        MoveL Target_3600,v30,fine,DrillTool\WObj:=FakeWing;
SetDO drillDone,1;
WaitUntil drillDone = 0;
        MoveL RelTool(Target_3600,0,0,-10),v30,z10,DrillTool\WObj:=FakeWing;
        MoveL RelTool(Target_3610,0,0,-10),v30,z10,DrillTool\WObj:=FakeWing;
        MoveL Target_3610,v30,fine,DrillTool\WObj:=FakeWing;
SetDO drillDone,1;
WaitUntil drillDone = 0;
        MoveL RelTool(Target_3610,0,0,-10),v30,z10,DrillTool\WObj:=FakeWing;
        MoveL RelTool(Target_3620,0,0,-10),v30,z10,DrillTool\WObj:=FakeWing;
        MoveL Target_3620,v30,fine,DrillTool\WObj:=FakeWing;
SetDO drillDone,1;
WaitUntil drillDone = 0;
        MoveL RelTool(Target_3620,0,0,-10),v30,z10,DrillTool\WObj:=FakeWing;
        MoveL RelTool(Target_3630,0,0,-10),v30,z10,DrillTool\WObj:=FakeWing;
        MoveL Target_3630,v30,fine,DrillTool\WObj:=FakeWing;
SetDO drillDone,1;
WaitUntil drillDone = 0;
        MoveL RelTool(Target_3630,0,0,-10),v30,z10,DrillTool\WObj:=FakeWing;
        MoveL RelTool(Target_3640,0,0,-10),v30,z10,DrillTool\WObj:=FakeWing;
        MoveL Target_3640,v30,fine,DrillTool\WObj:=FakeWing;
SetDO drillDone,1;
WaitUntil drillDone = 0;
        MoveL RelTool(Target_3640,0,0,-10),v30,z10,DrillTool\WObj:=FakeWing;
        MoveL RelTool(Target_3650,0,0,-10),v30,z10,DrillTool\WObj:=FakeWing;
        MoveL Target_3650,v30,fine,DrillTool\WObj:=FakeWing;
SetDO drillDone,1;
WaitUntil drillDone = 0;
        MoveL RelTool(Target_3650,0,0,-10),v30,z10,DrillTool\WObj:=FakeWing;
        MoveL RelTool(Target_3660,0,0,-10),v30,z10,DrillTool\WObj:=FakeWing;
        MoveL Target_3660,v30,fine,DrillTool\WObj:=FakeWing;
SetDO drillDone,1;
WaitUntil drillDone = 0;
        MoveL RelTool(Target_3660,0,0,-10),v30,z10,DrillTool\WObj:=FakeWing;
        MoveL RelTool(Target_3670,0,0,-10),v30,z10,DrillTool\WObj:=FakeWing;
        MoveL Target_3670,v30,fine,DrillTool\WObj:=FakeWing;
SetDO drillDone,1;
WaitUntil drillDone = 0;
        MoveL RelTool(Target_3670,0,0,-10),v30,z10,DrillTool\WObj:=FakeWing;
        MoveL RelTool(Target_3680,0,0,-10),v30,z10,DrillTool\WObj:=FakeWing;
        MoveL Target_3680,v30,fine,DrillTool\WObj:=FakeWing;
SetDO drillDone,1;
WaitUntil drillDone = 0;
        MoveL RelTool(Target_3680,0,0,-10),v30,z10,DrillTool\WObj:=FakeWing;
        MoveL RelTool(Target_3690,0,0,-10),v30,z10,DrillTool\WObj:=FakeWing;
        MoveL Target_3690,v30,fine,DrillTool\WObj:=FakeWing;
SetDO drillDone,1;
WaitUntil drillDone = 0;
        MoveL RelTool(Target_3690,0,0,-10),v30,z10,DrillTool\WObj:=FakeWing;
        MoveL RelTool(Target_3700,0,0,-10),v30,z10,DrillTool\WObj:=FakeWing;
        MoveL Target_3700,v30,fine,DrillTool\WObj:=FakeWing;
SetDO drillDone,1;
WaitUntil drillDone = 0;
        MoveL RelTool(Target_3700,0,0,-10),v30,z10,DrillTool\WObj:=FakeWing;
        MoveL RelTool(Target_3710,0,0,-10),v30,z10,DrillTool\WObj:=FakeWing;
        MoveL Target_3710,v30,fine,DrillTool\WObj:=FakeWing;
SetDO drillDone,1;
WaitUntil drillDone = 0;
        MoveL RelTool(Target_3710,0,0,-10),v30,z10,DrillTool\WObj:=FakeWing;
        MoveL RelTool(Target_3720,0,0,-10),v30,z10,DrillTool\WObj:=FakeWing;
        MoveL Target_3720,v30,fine,DrillTool\WObj:=FakeWing;
SetDO drillDone,1;
WaitUntil drillDone = 0;
        MoveL RelTool(Target_3720,0,0,-10),v30,z10,DrillTool\WObj:=FakeWing;
        MoveL RelTool(Target_3730,0,0,-10),v30,z10,DrillTool\WObj:=FakeWing;
        MoveL Target_3730,v30,fine,DrillTool\WObj:=FakeWing;
SetDO drillDone,1;
WaitUntil drillDone = 0;
        MoveL RelTool(Target_3730,0,0,-10),v30,z10,DrillTool\WObj:=FakeWing;
        MoveL RelTool(Target_3740,0,0,-10),v30,z10,DrillTool\WObj:=FakeWing;
        MoveL Target_3740,v30,fine,DrillTool\WObj:=FakeWing;
SetDO drillDone,1;
WaitUntil drillDone = 0;
        MoveL RelTool(Target_3740,0,0,-10),v30,z10,DrillTool\WObj:=FakeWing;
        MoveL RelTool(Target_3750,0,0,-10),v30,z10,DrillTool\WObj:=FakeWing;
        MoveL Target_3750,v30,fine,DrillTool\WObj:=FakeWing;
SetDO drillDone,1;
WaitUntil drillDone = 0;
        MoveL RelTool(Target_3750,0,0,-10),v30,z10,DrillTool\WObj:=FakeWing;
        MoveL RelTool(Target_3760,0,0,-10),v30,z10,DrillTool\WObj:=FakeWing;
        MoveL Target_3760,v30,fine,DrillTool\WObj:=FakeWing;
SetDO drillDone,1;
WaitUntil drillDone = 0;
        MoveL RelTool(Target_3760,0,0,-10),v30,z10,DrillTool\WObj:=FakeWing;
        MoveL RelTool(Target_3770,0,0,-10),v30,z10,DrillTool\WObj:=FakeWing;
        MoveL Target_3770,v30,fine,DrillTool\WObj:=FakeWing;
SetDO drillDone,1;
WaitUntil drillDone = 0;
        MoveL RelTool(Target_3770,0,0,-10),v30,z10,DrillTool\WObj:=FakeWing;
        MoveL RelTool(Target_3780,0,0,-10),v30,z10,DrillTool\WObj:=FakeWing;
        MoveL Target_3780,v30,fine,DrillTool\WObj:=FakeWing;
SetDO drillDone,1;
WaitUntil drillDone = 0;
        MoveL RelTool(Target_3780,0,0,-10),v30,z10,DrillTool\WObj:=FakeWing;
        MoveL RelTool(Target_3790,0,0,-10),v30,z10,DrillTool\WObj:=FakeWing;
        MoveL Target_3790,v30,fine,DrillTool\WObj:=FakeWing;
SetDO drillDone,1;
WaitUntil drillDone = 0;
        MoveL RelTool(Target_3790,0,0,-10),v30,z10,DrillTool\WObj:=FakeWing;
        MoveL RelTool(Target_3800,0,0,-10),v30,z10,DrillTool\WObj:=FakeWing;
        MoveL Target_3800,v30,fine,DrillTool\WObj:=FakeWing;
SetDO drillDone,1;
WaitUntil drillDone = 0;
        MoveL RelTool(Target_3800,0,0,-10),v30,z10,DrillTool\WObj:=FakeWing;
        MoveL RelTool(Target_3810,0,0,-10),v30,z10,DrillTool\WObj:=FakeWing;
        MoveL Target_3810,v30,fine,DrillTool\WObj:=FakeWing;
SetDO drillDone,1;
WaitUntil drillDone = 0;
        MoveL RelTool(Target_3810,0,0,-10),v30,z10,DrillTool\WObj:=FakeWing;
        MoveL RelTool(Target_3820,0,0,-10),v30,z10,DrillTool\WObj:=FakeWing;
        MoveL Target_3820,v30,fine,DrillTool\WObj:=FakeWing;
SetDO drillDone,1;
WaitUntil drillDone = 0;
        MoveL RelTool(Target_3820,0,0,-10),v30,z10,DrillTool\WObj:=FakeWing;
        MoveL RelTool(Target_3830,0,0,-10),v30,z10,DrillTool\WObj:=FakeWing;
        MoveL Target_3830,v30,fine,DrillTool\WObj:=FakeWing;
SetDO drillDone,1;
WaitUntil drillDone = 0;
        MoveL RelTool(Target_3830,0,0,-10),v30,z10,DrillTool\WObj:=FakeWing;
        MoveL RelTool(Target_3840,0,0,-10),v30,z10,DrillTool\WObj:=FakeWing;
        MoveL Target_3840,v30,fine,DrillTool\WObj:=FakeWing;
SetDO drillDone,1;
WaitUntil drillDone = 0;
        MoveL RelTool(Target_3840,0,0,-10),v30,z10,DrillTool\WObj:=FakeWing;
        MoveL RelTool(Target_3850,0,0,-10),v30,z10,DrillTool\WObj:=FakeWing;
        MoveL Target_3850,v30,fine,DrillTool\WObj:=FakeWing;
SetDO drillDone,1;
WaitUntil drillDone = 0;
        MoveL RelTool(Target_3850,0,0,-10),v30,z10,DrillTool\WObj:=FakeWing;
        MoveL RelTool(Target_3860,0,0,-10),v30,z10,DrillTool\WObj:=FakeWing;
        MoveL Target_3860,v30,fine,DrillTool\WObj:=FakeWing;
SetDO drillDone,1;
WaitUntil drillDone = 0;
        MoveL RelTool(Target_3860,0,0,-10),v30,z10,DrillTool\WObj:=FakeWing;
        MoveL RelTool(Target_3870,0,0,-10),v30,z10,DrillTool\WObj:=FakeWing;
        MoveL Target_3870,v30,fine,DrillTool\WObj:=FakeWing;
SetDO drillDone,1;
WaitUntil drillDone = 0;
        MoveL RelTool(Target_3870,0,0,-10),v30,z10,DrillTool\WObj:=FakeWing;
        MoveL RelTool(Target_3880,0,0,-10),v30,z10,DrillTool\WObj:=FakeWing;
        MoveL Target_3880,v30,fine,DrillTool\WObj:=FakeWing;
SetDO drillDone,1;
WaitUntil drillDone = 0;
        MoveL RelTool(Target_3880,0,0,-10),v30,z10,DrillTool\WObj:=FakeWing;
        MoveL RelTool(Target_3890,0,0,-10),v30,z10,DrillTool\WObj:=FakeWing;
        MoveL Target_3890,v30,fine,DrillTool\WObj:=FakeWing;
SetDO drillDone,1;
WaitUntil drillDone = 0;
        MoveL RelTool(Target_3890,0,0,-10),v30,z10,DrillTool\WObj:=FakeWing;
        MoveL RelTool(Target_3900,0,0,-10),v30,z10,DrillTool\WObj:=FakeWing;
        MoveL Target_3900,v30,fine,DrillTool\WObj:=FakeWing;
SetDO drillDone,1;
WaitUntil drillDone = 0;
        MoveL RelTool(Target_3900,0,0,-10),v30,z10,DrillTool\WObj:=FakeWing;
        MoveL RelTool(Target_3910,0,0,-10),v30,z10,DrillTool\WObj:=FakeWing;
        MoveL Target_3910,v30,fine,DrillTool\WObj:=FakeWing;
SetDO drillDone,1;
WaitUntil drillDone = 0;
        MoveL RelTool(Target_3910,0,0,-10),v30,z10,DrillTool\WObj:=FakeWing;
        MoveL RelTool(Target_3920,0,0,-10),v30,z10,DrillTool\WObj:=FakeWing;
        MoveL Target_3920,v30,fine,DrillTool\WObj:=FakeWing;
SetDO drillDone,1;
WaitUntil drillDone = 0;
        MoveL RelTool(Target_3920,0,0,-10),v30,z10,DrillTool\WObj:=FakeWing;
        MoveL RelTool(Target_3930,0,0,-10),v30,z10,DrillTool\WObj:=FakeWing;
        MoveL Target_3930,v30,fine,DrillTool\WObj:=FakeWing;
SetDO drillDone,1;
WaitUntil drillDone = 0;
        MoveL RelTool(Target_3930,0,0,-10),v30,z10,DrillTool\WObj:=FakeWing;
        MoveL RelTool(Target_3940,0,0,-10),v30,z10,DrillTool\WObj:=FakeWing;
        MoveL Target_3940,v30,fine,DrillTool\WObj:=FakeWing;
SetDO drillDone,1;
WaitUntil drillDone = 0;
        MoveL RelTool(Target_3940,0,0,-10),v30,z10,DrillTool\WObj:=FakeWing;
        MoveL RelTool(Target_3950,0,0,-10),v30,z10,DrillTool\WObj:=FakeWing;
        MoveL Target_3950,v30,fine,DrillTool\WObj:=FakeWing;
SetDO drillDone,1;
WaitUntil drillDone = 0;
        MoveL RelTool(Target_3950,0,0,-10),v30,z10,DrillTool\WObj:=FakeWing;
        MoveL RelTool(Target_3960,0,0,-10),v30,z10,DrillTool\WObj:=FakeWing;
        MoveL Target_3960,v30,fine,DrillTool\WObj:=FakeWing;
SetDO drillDone,1;
WaitUntil drillDone = 0;
        MoveL RelTool(Target_3960,0,0,-10),v30,z10,DrillTool\WObj:=FakeWing;
        MoveL RelTool(Target_3970,0,0,-10),v30,z10,DrillTool\WObj:=FakeWing;
        MoveL Target_3970,v30,fine,DrillTool\WObj:=FakeWing;
SetDO drillDone,1;
WaitUntil drillDone = 0;
        MoveL RelTool(Target_3970,0,0,-10),v30,z10,DrillTool\WObj:=FakeWing;
        MoveL RelTool(Target_3980,0,0,-10),v30,z10,DrillTool\WObj:=FakeWing;
        MoveL Target_3980,v30,fine,DrillTool\WObj:=FakeWing;
SetDO drillDone,1;
WaitUntil drillDone = 0;
        MoveL RelTool(Target_3980,0,0,-10),v30,z10,DrillTool\WObj:=FakeWing;
        MoveL RelTool(Target_3990,0,0,-10),v30,z10,DrillTool\WObj:=FakeWing;
        MoveL Target_3990,v30,fine,DrillTool\WObj:=FakeWing;
SetDO drillDone,1;
WaitUntil drillDone = 0;
        MoveL RelTool(Target_3990,0,0,-10),v30,z10,DrillTool\WObj:=FakeWing;
        MoveL RelTool(Target_4000,0,0,-10),v30,z10,DrillTool\WObj:=FakeWing;
        MoveL Target_4000,v30,fine,DrillTool\WObj:=FakeWing;
SetDO drillDone,1;
WaitUntil drillDone = 0;
        MoveL RelTool(Target_4000,0,0,-10),v30,z10,DrillTool\WObj:=FakeWing;
        MoveL RelTool(Target_4010,0,0,-10),v30,z10,DrillTool\WObj:=FakeWing;
        MoveL Target_4010,v30,fine,DrillTool\WObj:=FakeWing;
SetDO drillDone,1;
WaitUntil drillDone = 0;
        MoveL RelTool(Target_4010,0,0,-10),v30,z10,DrillTool\WObj:=FakeWing;
        MoveL RelTool(Target_4020,0,0,-10),v30,z10,DrillTool\WObj:=FakeWing;
        MoveL Target_4020,v30,fine,DrillTool\WObj:=FakeWing;
SetDO drillDone,1;
WaitUntil drillDone = 0;
        MoveL RelTool(Target_4020,0,0,-10),v30,z10,DrillTool\WObj:=FakeWing;
        MoveL RelTool(Target_4030,0,0,-10),v30,z10,DrillTool\WObj:=FakeWing;
        MoveL Target_4030,v30,fine,DrillTool\WObj:=FakeWing;
SetDO drillDone,1;
WaitUntil drillDone = 0;
        MoveL RelTool(Target_4030,0,0,-10),v30,z10,DrillTool\WObj:=FakeWing;
        MoveL RelTool(Target_4040,0,0,-10),v30,z10,DrillTool\WObj:=FakeWing;
        MoveL Target_4040,v30,fine,DrillTool\WObj:=FakeWing;
SetDO drillDone,1;
WaitUntil drillDone = 0;
        MoveL RelTool(Target_4040,0,0,-10),v30,z10,DrillTool\WObj:=FakeWing;
        MoveL RelTool(Target_4050,0,0,-10),v30,z10,DrillTool\WObj:=FakeWing;
        MoveL Target_4050,v30,fine,DrillTool\WObj:=FakeWing;
SetDO drillDone,1;
WaitUntil drillDone = 0;
        MoveL RelTool(Target_4050,0,0,-10),v30,z10,DrillTool\WObj:=FakeWing;
        MoveL RelTool(Target_4060,0,0,-10),v30,z10,DrillTool\WObj:=FakeWing;
        MoveL Target_4060,v30,fine,DrillTool\WObj:=FakeWing;
SetDO drillDone,1;
WaitUntil drillDone = 0;
        MoveL RelTool(Target_4060,0,0,-10),v30,z10,DrillTool\WObj:=FakeWing;
        MoveL RelTool(Target_4070,0,0,-10),v30,z10,DrillTool\WObj:=FakeWing;
        MoveL Target_4070,v30,fine,DrillTool\WObj:=FakeWing;
SetDO drillDone,1;
WaitUntil drillDone = 0;
        MoveL RelTool(Target_4070,0,0,-10),v30,z10,DrillTool\WObj:=FakeWing;
        MoveL RelTool(Target_4080,0,0,-10),v30,z10,DrillTool\WObj:=FakeWing;
        MoveL Target_4080,v30,fine,DrillTool\WObj:=FakeWing;
SetDO drillDone,1;
WaitUntil drillDone = 0;
        MoveL RelTool(Target_4080,0,0,-10),v30,z10,DrillTool\WObj:=FakeWing;
        MoveL RelTool(Target_4090,0,0,-10),v30,z10,DrillTool\WObj:=FakeWing;
        MoveL Target_4090,v30,fine,DrillTool\WObj:=FakeWing;
SetDO drillDone,1;
WaitUntil drillDone = 0;
        MoveL RelTool(Target_4090,0,0,-10),v30,z10,DrillTool\WObj:=FakeWing;
        MoveL RelTool(Target_4100,0,0,-10),v30,z10,DrillTool\WObj:=FakeWing;
        MoveL Target_4100,v30,fine,DrillTool\WObj:=FakeWing;
SetDO drillDone,1;
WaitUntil drillDone = 0;
        MoveL RelTool(Target_4100,0,0,-10),v30,z10,DrillTool\WObj:=FakeWing;
        MoveL RelTool(Target_4110,0,0,-10),v30,z10,DrillTool\WObj:=FakeWing;
        MoveL Target_4110,v30,fine,DrillTool\WObj:=FakeWing;
SetDO drillDone,1;
WaitUntil drillDone = 0;
        MoveL RelTool(Target_4110,0,0,-10),v30,z10,DrillTool\WObj:=FakeWing;
        MoveL RelTool(Target_4120,0,0,-10),v30,z10,DrillTool\WObj:=FakeWing;
        MoveL Target_4120,v30,fine,DrillTool\WObj:=FakeWing;
SetDO drillDone,1;
WaitUntil drillDone = 0;
        MoveL RelTool(Target_4120,0,0,-10),v30,z10,DrillTool\WObj:=FakeWing;
        MoveL RelTool(Target_4130,0,0,-10),v30,z10,DrillTool\WObj:=FakeWing;
        MoveL Target_4130,v30,fine,DrillTool\WObj:=FakeWing;
SetDO drillDone,1;
WaitUntil drillDone = 0;
        MoveL RelTool(Target_4130,0,0,-10),v30,z10,DrillTool\WObj:=FakeWing;
        MoveL RelTool(Target_4140,0,0,-10),v30,z10,DrillTool\WObj:=FakeWing;
        MoveL Target_4140,v30,fine,DrillTool\WObj:=FakeWing;
SetDO drillDone,1;
WaitUntil drillDone = 0;
        MoveL RelTool(Target_4140,0,0,-10),v30,z10,DrillTool\WObj:=FakeWing;
        MoveL RelTool(Target_4150,0,0,-10),v30,z10,DrillTool\WObj:=FakeWing;
        MoveL Target_4150,v30,fine,DrillTool\WObj:=FakeWing;
SetDO drillDone,1;
WaitUntil drillDone = 0;
        MoveL RelTool(Target_4150,0,0,-10),v30,z10,DrillTool\WObj:=FakeWing;
        MoveL RelTool(Target_4160,0,0,-10),v30,z10,DrillTool\WObj:=FakeWing;
        MoveL Target_4160,v30,fine,DrillTool\WObj:=FakeWing;
SetDO drillDone,1;
WaitUntil drillDone = 0;
        MoveL RelTool(Target_4160,0,0,-10),v30,z10,DrillTool\WObj:=FakeWing;
        MoveL RelTool(Target_4170,0,0,-10),v30,z10,DrillTool\WObj:=FakeWing;
        MoveL Target_4170,v30,fine,DrillTool\WObj:=FakeWing;
SetDO drillDone,1;
WaitUntil drillDone = 0;
        MoveL RelTool(Target_4170,0,0,-10),v30,z10,DrillTool\WObj:=FakeWing;
        MoveL RelTool(Target_4180,0,0,-10),v30,z10,DrillTool\WObj:=FakeWing;
        MoveL Target_4180,v30,fine,DrillTool\WObj:=FakeWing;
SetDO drillDone,1;
WaitUntil drillDone = 0;
        MoveL RelTool(Target_4180,0,0,-10),v30,z10,DrillTool\WObj:=FakeWing;
        MoveL RelTool(Target_4190,0,0,-10),v30,z10,DrillTool\WObj:=FakeWing;
        MoveL Target_4190,v30,fine,DrillTool\WObj:=FakeWing;
SetDO drillDone,1;
WaitUntil drillDone = 0;
        MoveL RelTool(Target_4190,0,0,-10),v30,z10,DrillTool\WObj:=FakeWing;
        MoveL RelTool(Target_4200,0,0,-10),v30,z10,DrillTool\WObj:=FakeWing;
        MoveL Target_4200,v30,fine,DrillTool\WObj:=FakeWing;
SetDO drillDone,1;
WaitUntil drillDone = 0;
        MoveL RelTool(Target_4200,0,0,-10),v30,z10,DrillTool\WObj:=FakeWing;
        MoveL RelTool(Target_4210,0,0,-10),v30,z10,DrillTool\WObj:=FakeWing;
        MoveL Target_4210,v30,fine,DrillTool\WObj:=FakeWing;
SetDO drillDone,1;
WaitUntil drillDone = 0;
        MoveL RelTool(Target_4210,0,0,-10),v30,z10,DrillTool\WObj:=FakeWing;
        MoveL RelTool(Target_4220,0,0,-10),v30,z10,DrillTool\WObj:=FakeWing;
        MoveL Target_4220,v30,fine,DrillTool\WObj:=FakeWing;
SetDO drillDone,1;
WaitUntil drillDone = 0;
        MoveL RelTool(Target_4220,0,0,-10),v30,z10,DrillTool\WObj:=FakeWing;
        MoveL RelTool(Target_4230,0,0,-10),v30,z10,DrillTool\WObj:=FakeWing;
        MoveL Target_4230,v30,fine,DrillTool\WObj:=FakeWing;
SetDO drillDone,1;
WaitUntil drillDone = 0;
        MoveL RelTool(Target_4230,0,0,-10),v30,z10,DrillTool\WObj:=FakeWing;
        MoveL RelTool(Target_4240,0,0,-10),v30,z10,DrillTool\WObj:=FakeWing;
        MoveL Target_4240,v30,fine,DrillTool\WObj:=FakeWing;
SetDO drillDone,1;
WaitUntil drillDone = 0;
        MoveL RelTool(Target_4240,0,0,-10),v30,z10,DrillTool\WObj:=FakeWing;
        MoveL RelTool(Target_4250,0,0,-10),v30,z10,DrillTool\WObj:=FakeWing;
        MoveL Target_4250,v30,fine,DrillTool\WObj:=FakeWing;
SetDO drillDone,1;
WaitUntil drillDone = 0;
        MoveL RelTool(Target_4250,0,0,-10),v30,z10,DrillTool\WObj:=FakeWing;
        MoveL RelTool(Target_4260,0,0,-10),v30,z10,DrillTool\WObj:=FakeWing;
        MoveL Target_4260,v30,fine,DrillTool\WObj:=FakeWing;
SetDO drillDone,1;
WaitUntil drillDone = 0;
        MoveL RelTool(Target_4260,0,0,-10),v30,z10,DrillTool\WObj:=FakeWing;
        MoveL RelTool(Target_4270,0,0,-10),v30,z10,DrillTool\WObj:=FakeWing;
        MoveL Target_4270,v30,fine,DrillTool\WObj:=FakeWing;
SetDO drillDone,1;
WaitUntil drillDone = 0;
        MoveL RelTool(Target_4270,0,0,-10),v30,z10,DrillTool\WObj:=FakeWing;
        MoveL RelTool(Target_4280,0,0,-10),v30,z10,DrillTool\WObj:=FakeWing;
        MoveL Target_4280,v30,fine,DrillTool\WObj:=FakeWing;
SetDO drillDone,1;
WaitUntil drillDone = 0;
        MoveL RelTool(Target_4280,0,0,-10),v30,z10,DrillTool\WObj:=FakeWing;
        MoveL RelTool(Target_4290,0,0,-10),v30,z10,DrillTool\WObj:=FakeWing;
        MoveL Target_4290,v30,fine,DrillTool\WObj:=FakeWing;
SetDO drillDone,1;
WaitUntil drillDone = 0;
        MoveL RelTool(Target_4290,0,0,-10),v30,z10,DrillTool\WObj:=FakeWing;
        MoveL RelTool(Target_4300,0,0,-10),v30,z10,DrillTool\WObj:=FakeWing;
        MoveL Target_4300,v30,fine,DrillTool\WObj:=FakeWing;
SetDO drillDone,1;
WaitUntil drillDone = 0;
        MoveL RelTool(Target_4300,0,0,-10),v30,z10,DrillTool\WObj:=FakeWing;
        MoveL RelTool(Target_4310,0,0,-10),v30,z10,DrillTool\WObj:=FakeWing;
        MoveL Target_4310,v30,fine,DrillTool\WObj:=FakeWing;
SetDO drillDone,1;
WaitUntil drillDone = 0;
        MoveL RelTool(Target_4310,0,0,-10),v30,z10,DrillTool\WObj:=FakeWing;
        MoveL RelTool(Target_4320,0,0,-10),v30,z10,DrillTool\WObj:=FakeWing;
        MoveL Target_4320,v30,fine,DrillTool\WObj:=FakeWing;
SetDO drillDone,1;
WaitUntil drillDone = 0;
        MoveL RelTool(Target_4320,0,0,-10),v30,z10,DrillTool\WObj:=FakeWing;
        MoveL RelTool(Target_4330,0,0,-10),v30,z10,DrillTool\WObj:=FakeWing;
        MoveL Target_4330,v30,fine,DrillTool\WObj:=FakeWing;
SetDO drillDone,1;
WaitUntil drillDone = 0;
        MoveL RelTool(Target_4330,0,0,-10),v30,z10,DrillTool\WObj:=FakeWing;
        MoveL RelTool(Target_4340,0,0,-10),v30,z10,DrillTool\WObj:=FakeWing;
        MoveL Target_4340,v30,fine,DrillTool\WObj:=FakeWing;
SetDO drillDone,1;
WaitUntil drillDone = 0;
        MoveL RelTool(Target_4340,0,0,-10),v30,z10,DrillTool\WObj:=FakeWing;
        MoveL RelTool(Target_4350,0,0,-10),v30,z10,DrillTool\WObj:=FakeWing;
        MoveL Target_4350,v30,fine,DrillTool\WObj:=FakeWing;
SetDO drillDone,1;
WaitUntil drillDone = 0;
        MoveL RelTool(Target_4350,0,0,-10),v30,z10,DrillTool\WObj:=FakeWing;
        MoveL RelTool(Target_4360,0,0,-10),v30,z10,DrillTool\WObj:=FakeWing;
        MoveL Target_4360,v30,fine,DrillTool\WObj:=FakeWing;
SetDO drillDone,1;
WaitUntil drillDone = 0;
        MoveL RelTool(Target_4360,0,0,-10),v30,z10,DrillTool\WObj:=FakeWing;
        MoveL RelTool(Target_4370,0,0,-10),v30,z10,DrillTool\WObj:=FakeWing;
        MoveL Target_4370,v30,fine,DrillTool\WObj:=FakeWing;
SetDO drillDone,1;
WaitUntil drillDone = 0;
        MoveL RelTool(Target_4370,0,0,-10),v30,z10,DrillTool\WObj:=FakeWing;
        MoveL RelTool(Target_4380,0,0,-10),v30,z10,DrillTool\WObj:=FakeWing;
        MoveL Target_4380,v30,fine,DrillTool\WObj:=FakeWing;
SetDO drillDone,1;
WaitUntil drillDone = 0;
        MoveL RelTool(Target_4380,0,0,-10),v30,z10,DrillTool\WObj:=FakeWing;
        MoveL RelTool(Target_4390,0,0,-10),v30,z10,DrillTool\WObj:=FakeWing;
        MoveL Target_4390,v30,fine,DrillTool\WObj:=FakeWing;
SetDO drillDone,1;
WaitUntil drillDone = 0;
        MoveL RelTool(Target_4390,0,0,-10),v30,z10,DrillTool\WObj:=FakeWing;
        MoveL RelTool(Target_4400,0,0,-10),v30,z10,DrillTool\WObj:=FakeWing;
        MoveL Target_4400,v30,fine,DrillTool\WObj:=FakeWing;
SetDO drillDone,1;
WaitUntil drillDone = 0;
        MoveL RelTool(Target_4400,0,0,-10),v30,z10,DrillTool\WObj:=FakeWing;
        MoveL RelTool(Target_4410,0,0,-10),v30,z10,DrillTool\WObj:=FakeWing;
        MoveL Target_4410,v30,fine,DrillTool\WObj:=FakeWing;
SetDO drillDone,1;
WaitUntil drillDone = 0;
        MoveL RelTool(Target_4410,0,0,-10),v30,z10,DrillTool\WObj:=FakeWing;
        MoveL RelTool(Target_4420,0,0,-10),v30,z10,DrillTool\WObj:=FakeWing;
        MoveL Target_4420,v30,fine,DrillTool\WObj:=FakeWing;
SetDO drillDone,1;
WaitUntil drillDone = 0;
        MoveL RelTool(Target_4420,0,0,-10),v30,z10,DrillTool\WObj:=FakeWing;
        MoveL RelTool(Target_4430,0,0,-10),v30,z10,DrillTool\WObj:=FakeWing;
        MoveL Target_4430,v30,fine,DrillTool\WObj:=FakeWing;
SetDO drillDone,1;
WaitUntil drillDone = 0;
        MoveL RelTool(Target_4430,0,0,-10),v30,z10,DrillTool\WObj:=FakeWing;
        MoveL RelTool(Target_4440,0,0,-10),v30,z10,DrillTool\WObj:=FakeWing;
        MoveL Target_4440,v30,fine,DrillTool\WObj:=FakeWing;
SetDO drillDone,1;
WaitUntil drillDone = 0;
        MoveL RelTool(Target_4440,0,0,-10),v30,z10,DrillTool\WObj:=FakeWing;
        MoveL RelTool(Target_4450,0,0,-10),v30,z10,DrillTool\WObj:=FakeWing;
        MoveL Target_4450,v30,fine,DrillTool\WObj:=FakeWing;
SetDO drillDone,1;
WaitUntil drillDone = 0;
        MoveL RelTool(Target_4450,0,0,-10),v30,z10,DrillTool\WObj:=FakeWing;
        MoveL RelTool(Target_4460,0,0,-10),v30,z10,DrillTool\WObj:=FakeWing;
        MoveL Target_4460,v30,fine,DrillTool\WObj:=FakeWing;
SetDO drillDone,1;
WaitUntil drillDone = 0;
        MoveL RelTool(Target_4460,0,0,-10),v30,z10,DrillTool\WObj:=FakeWing;
        MoveL RelTool(Target_4470,0,0,-10),v30,z10,DrillTool\WObj:=FakeWing;
        MoveL Target_4470,v30,fine,DrillTool\WObj:=FakeWing;
SetDO drillDone,1;
WaitUntil drillDone = 0;
        MoveL RelTool(Target_4470,0,0,-10),v30,z10,DrillTool\WObj:=FakeWing;
        MoveL RelTool(Target_4480,0,0,-10),v30,z10,DrillTool\WObj:=FakeWing;
        MoveL Target_4480,v30,fine,DrillTool\WObj:=FakeWing;
SetDO drillDone,1;
WaitUntil drillDone = 0;
        MoveL RelTool(Target_4480,0,0,-10),v30,z10,DrillTool\WObj:=FakeWing;
        MoveL RelTool(Target_4490,0,0,-10),v30,z10,DrillTool\WObj:=FakeWing;
        MoveL Target_4490,v30,fine,DrillTool\WObj:=FakeWing;
SetDO drillDone,1;
WaitUntil drillDone = 0;
        MoveL RelTool(Target_4490,0,0,-10),v30,z10,DrillTool\WObj:=FakeWing;
        MoveL RelTool(Target_4500,0,0,-10),v30,z10,DrillTool\WObj:=FakeWing;
        MoveL Target_4500,v30,fine,DrillTool\WObj:=FakeWing;
SetDO drillDone,1;
WaitUntil drillDone = 0;
        MoveL RelTool(Target_4500,0,0,-10),v30,z10,DrillTool\WObj:=FakeWing;
        MoveL RelTool(Target_4510,0,0,-10),v30,z10,DrillTool\WObj:=FakeWing;
        MoveL Target_4510,v30,fine,DrillTool\WObj:=FakeWing;
SetDO drillDone,1;
WaitUntil drillDone = 0;
        MoveL RelTool(Target_4510,0,0,-10),v30,z10,DrillTool\WObj:=FakeWing;
        MoveL RelTool(Target_4520,0,0,-10),v30,z10,DrillTool\WObj:=FakeWing;
        MoveL Target_4520,v30,fine,DrillTool\WObj:=FakeWing;
SetDO drillDone,1;
WaitUntil drillDone = 0;
        MoveL RelTool(Target_4520,0,0,-10),v30,z10,DrillTool\WObj:=FakeWing;
        MoveL RelTool(Target_4530,0,0,-10),v30,z10,DrillTool\WObj:=FakeWing;
        MoveL Target_4530,v30,fine,DrillTool\WObj:=FakeWing;
SetDO drillDone,1;
WaitUntil drillDone = 0;
        MoveL RelTool(Target_4530,0,0,-10),v30,z10,DrillTool\WObj:=FakeWing;
        MoveL RelTool(Target_4540,0,0,-10),v30,z10,DrillTool\WObj:=FakeWing;
        MoveL Target_4540,v30,fine,DrillTool\WObj:=FakeWing;
SetDO drillDone,1;
WaitUntil drillDone = 0;
        MoveL RelTool(Target_4540,0,0,-10),v30,z10,DrillTool\WObj:=FakeWing;
        MoveL RelTool(Target_4550,0,0,-10),v30,z10,DrillTool\WObj:=FakeWing;
        MoveL Target_4550,v30,fine,DrillTool\WObj:=FakeWing;
SetDO drillDone,1;
WaitUntil drillDone = 0;
        MoveL RelTool(Target_4550,0,0,-10),v30,z10,DrillTool\WObj:=FakeWing;
        MoveL RelTool(Target_4560,0,0,-10),v30,z10,DrillTool\WObj:=FakeWing;
        MoveL Target_4560,v30,fine,DrillTool\WObj:=FakeWing;
SetDO drillDone,1;
WaitUntil drillDone = 0;
        MoveL RelTool(Target_4560,0,0,-10),v30,z10,DrillTool\WObj:=FakeWing;
        MoveL RelTool(Target_4570,0,0,-10),v30,z10,DrillTool\WObj:=FakeWing;
        MoveL Target_4570,v30,fine,DrillTool\WObj:=FakeWing;
SetDO drillDone,1;
WaitUntil drillDone = 0;
        MoveL RelTool(Target_4570,0,0,-10),v30,z10,DrillTool\WObj:=FakeWing;
        MoveL RelTool(Target_4580,0,0,-10),v30,z10,DrillTool\WObj:=FakeWing;
        MoveL Target_4580,v30,fine,DrillTool\WObj:=FakeWing;
SetDO drillDone,1;
WaitUntil drillDone = 0;
        MoveL RelTool(Target_4580,0,0,-10),v30,z10,DrillTool\WObj:=FakeWing;
        MoveL RelTool(Target_4590,0,0,-10),v30,z10,DrillTool\WObj:=FakeWing;
        MoveL Target_4590,v30,fine,DrillTool\WObj:=FakeWing;
SetDO drillDone,1;
WaitUntil drillDone = 0;
        MoveL RelTool(Target_4590,0,0,-10),v30,z10,DrillTool\WObj:=FakeWing;
        MoveL RelTool(Target_4600,0,0,-10),v30,z10,DrillTool\WObj:=FakeWing;
        MoveL Target_4600,v30,fine,DrillTool\WObj:=FakeWing;
SetDO drillDone,1;
WaitUntil drillDone = 0;
        MoveL RelTool(Target_4600,0,0,-10),v30,z10,DrillTool\WObj:=FakeWing;
        MoveL RelTool(Target_4610,0,0,-10),v30,z10,DrillTool\WObj:=FakeWing;
        MoveL Target_4610,v30,fine,DrillTool\WObj:=FakeWing;
SetDO drillDone,1;
WaitUntil drillDone = 0;
        MoveL RelTool(Target_4610,0,0,-10),v30,z10,DrillTool\WObj:=FakeWing;
        MoveL RelTool(Target_4620,0,0,-10),v30,z10,DrillTool\WObj:=FakeWing;
        MoveL Target_4620,v30,fine,DrillTool\WObj:=FakeWing;
SetDO drillDone,1;
WaitUntil drillDone = 0;
        MoveL RelTool(Target_4620,0,0,-10),v30,z10,DrillTool\WObj:=FakeWing;
        MoveL RelTool(Target_4630,0,0,-10),v30,z10,DrillTool\WObj:=FakeWing;
        MoveL Target_4630,v30,fine,DrillTool\WObj:=FakeWing;
SetDO drillDone,1;
WaitUntil drillDone = 0;
        MoveL RelTool(Target_4630,0,0,-10),v30,z10,DrillTool\WObj:=FakeWing;
        MoveL RelTool(Target_4640,0,0,-10),v30,z10,DrillTool\WObj:=FakeWing;
        MoveL Target_4640,v30,fine,DrillTool\WObj:=FakeWing;
SetDO drillDone,1;
WaitUntil drillDone = 0;
        MoveL RelTool(Target_4640,0,0,-10),v30,z10,DrillTool\WObj:=FakeWing;
        MoveL RelTool(Target_4650,0,0,-10),v30,z10,DrillTool\WObj:=FakeWing;
        MoveL Target_4650,v30,fine,DrillTool\WObj:=FakeWing;
SetDO drillDone,1;
WaitUntil drillDone = 0;
        MoveL RelTool(Target_4650,0,0,-10),v30,z10,DrillTool\WObj:=FakeWing;
        MoveL RelTool(Target_4660,0,0,-10),v30,z10,DrillTool\WObj:=FakeWing;
        MoveL Target_4660,v30,fine,DrillTool\WObj:=FakeWing;
SetDO drillDone,1;
WaitUntil drillDone = 0;
        MoveL RelTool(Target_4660,0,0,-10),v30,z10,DrillTool\WObj:=FakeWing;
        MoveL RelTool(Target_4670,0,0,-10),v30,z10,DrillTool\WObj:=FakeWing;
        MoveL Target_4670,v30,fine,DrillTool\WObj:=FakeWing;
SetDO drillDone,1;
WaitUntil drillDone = 0;
        MoveL RelTool(Target_4670,0,0,-10),v30,z10,DrillTool\WObj:=FakeWing;
        MoveL RelTool(Target_4680,0,0,-10),v30,z10,DrillTool\WObj:=FakeWing;
        MoveL Target_4680,v30,fine,DrillTool\WObj:=FakeWing;
SetDO drillDone,1;
WaitUntil drillDone = 0;
        MoveL RelTool(Target_4680,0,0,-10),v30,z10,DrillTool\WObj:=FakeWing;
        MoveL RelTool(Target_4690,0,0,-10),v30,z10,DrillTool\WObj:=FakeWing;
        MoveL Target_4690,v30,fine,DrillTool\WObj:=FakeWing;
SetDO drillDone,1;
WaitUntil drillDone = 0;
        MoveL RelTool(Target_4690,0,0,-10),v30,z10,DrillTool\WObj:=FakeWing;
        MoveL RelTool(Target_4700,0,0,-10),v30,z10,DrillTool\WObj:=FakeWing;
        MoveL Target_4700,v30,fine,DrillTool\WObj:=FakeWing;
SetDO drillDone,1;
WaitUntil drillDone = 0;
        MoveL RelTool(Target_4700,0,0,-10),v30,z10,DrillTool\WObj:=FakeWing;
        MoveL RelTool(Target_4710,0,0,-10),v30,z10,DrillTool\WObj:=FakeWing;
        MoveL Target_4710,v30,fine,DrillTool\WObj:=FakeWing;
SetDO drillDone,1;
WaitUntil drillDone = 0;
        MoveL RelTool(Target_4710,0,0,-10),v30,z10,DrillTool\WObj:=FakeWing;
        MoveL RelTool(Target_4720,0,0,-10),v30,z10,DrillTool\WObj:=FakeWing;
        MoveL Target_4720,v30,fine,DrillTool\WObj:=FakeWing;
SetDO drillDone,1;
WaitUntil drillDone = 0;
        MoveL RelTool(Target_4720,0,0,-10),v30,z10,DrillTool\WObj:=FakeWing;
        MoveL RelTool(Target_4730,0,0,-10),v30,z10,DrillTool\WObj:=FakeWing;
        MoveL Target_4730,v30,fine,DrillTool\WObj:=FakeWing;
SetDO drillDone,1;
WaitUntil drillDone = 0;
        MoveL RelTool(Target_4730,0,0,-10),v30,z10,DrillTool\WObj:=FakeWing;
        MoveL RelTool(Target_4740,0,0,-10),v30,z10,DrillTool\WObj:=FakeWing;
        MoveL Target_4740,v30,fine,DrillTool\WObj:=FakeWing;
SetDO drillDone,1;
WaitUntil drillDone = 0;
        MoveL RelTool(Target_4740,0,0,-10),v30,z10,DrillTool\WObj:=FakeWing;
        MoveL RelTool(Target_4750,0,0,-10),v30,z10,DrillTool\WObj:=FakeWing;
        MoveL Target_4750,v30,fine,DrillTool\WObj:=FakeWing;
SetDO drillDone,1;
WaitUntil drillDone = 0;
        MoveL RelTool(Target_4750,0,0,-10),v30,z10,DrillTool\WObj:=FakeWing;
        MoveL RelTool(Target_4760,0,0,-10),v30,z10,DrillTool\WObj:=FakeWing;
        MoveL Target_4760,v30,fine,DrillTool\WObj:=FakeWing;
SetDO drillDone,1;
WaitUntil drillDone = 0;
        MoveL RelTool(Target_4760,0,0,-10),v30,z10,DrillTool\WObj:=FakeWing;
        MoveL RelTool(Target_4770,0,0,-10),v30,z10,DrillTool\WObj:=FakeWing;
        MoveL Target_4770,v30,fine,DrillTool\WObj:=FakeWing;
SetDO drillDone,1;
WaitUntil drillDone = 0;
        MoveL RelTool(Target_4770,0,0,-10),v30,z10,DrillTool\WObj:=FakeWing;
        MoveL RelTool(Target_4780,0,0,-10),v30,z10,DrillTool\WObj:=FakeWing;
        MoveL Target_4780,v30,fine,DrillTool\WObj:=FakeWing;
SetDO drillDone,1;
WaitUntil drillDone = 0;
        MoveL RelTool(Target_4780,0,0,-10),v30,z10,DrillTool\WObj:=FakeWing;
        MoveL RelTool(Target_4790,0,0,-10),v30,z10,DrillTool\WObj:=FakeWing;
        MoveL Target_4790,v30,fine,DrillTool\WObj:=FakeWing;
SetDO drillDone,1;
WaitUntil drillDone = 0;
        MoveL RelTool(Target_4790,0,0,-10),v30,z10,DrillTool\WObj:=FakeWing;
        MoveL RelTool(Target_4800,0,0,-10),v30,z10,DrillTool\WObj:=FakeWing;
        MoveL Target_4800,v30,fine,DrillTool\WObj:=FakeWing;
SetDO drillDone,1;
WaitUntil drillDone = 0;
        MoveL RelTool(Target_4800,0,0,-10),v30,z10,DrillTool\WObj:=FakeWing;
        MoveL RelTool(Target_4810,0,0,-10),v30,z10,DrillTool\WObj:=FakeWing;
        MoveL Target_4810,v30,fine,DrillTool\WObj:=FakeWing;
SetDO drillDone,1;
WaitUntil drillDone = 0;
        MoveL RelTool(Target_4810,0,0,-10),v30,z10,DrillTool\WObj:=FakeWing;
        MoveL RelTool(Target_4820,0,0,-10),v30,z10,DrillTool\WObj:=FakeWing;
        MoveL Target_4820,v30,fine,DrillTool\WObj:=FakeWing;
SetDO drillDone,1;
WaitUntil drillDone = 0;
        MoveL RelTool(Target_4820,0,0,-10),v30,z10,DrillTool\WObj:=FakeWing;
        MoveL RelTool(Target_4830,0,0,-10),v30,z10,DrillTool\WObj:=FakeWing;
        MoveL Target_4830,v30,fine,DrillTool\WObj:=FakeWing;
SetDO drillDone,1;
WaitUntil drillDone = 0;
        MoveL RelTool(Target_4830,0,0,-10),v30,z10,DrillTool\WObj:=FakeWing;
        MoveL RelTool(Target_4840,0,0,-10),v30,z10,DrillTool\WObj:=FakeWing;
        MoveL Target_4840,v30,fine,DrillTool\WObj:=FakeWing;
SetDO drillDone,1;
WaitUntil drillDone = 0;
        MoveL RelTool(Target_4840,0,0,-10),v30,z10,DrillTool\WObj:=FakeWing;
        MoveL RelTool(Target_4850,0,0,-10),v30,z10,DrillTool\WObj:=FakeWing;
        MoveL Target_4850,v30,fine,DrillTool\WObj:=FakeWing;
SetDO drillDone,1;
WaitUntil drillDone = 0;
        MoveL RelTool(Target_4850,0,0,-10),v30,z10,DrillTool\WObj:=FakeWing;
        MoveL RelTool(Target_4860,0,0,-10),v30,z10,DrillTool\WObj:=FakeWing;
        MoveL Target_4860,v30,fine,DrillTool\WObj:=FakeWing;
SetDO drillDone,1;
WaitUntil drillDone = 0;
        MoveL RelTool(Target_4860,0,0,-10),v30,z10,DrillTool\WObj:=FakeWing;
        MoveL RelTool(Target_4870,0,0,-10),v30,z10,DrillTool\WObj:=FakeWing;
        MoveL Target_4870,v30,fine,DrillTool\WObj:=FakeWing;
SetDO drillDone,1;
WaitUntil drillDone = 0;
        MoveL RelTool(Target_4870,0,0,-10),v30,z10,DrillTool\WObj:=FakeWing;
        MoveL RelTool(Target_4880,0,0,-10),v30,z10,DrillTool\WObj:=FakeWing;
        MoveL Target_4880,v30,fine,DrillTool\WObj:=FakeWing;
SetDO drillDone,1;
WaitUntil drillDone = 0;
        MoveL RelTool(Target_4880,0,0,-10),v30,z10,DrillTool\WObj:=FakeWing;
        MoveL RelTool(Target_4890,0,0,-10),v30,z10,DrillTool\WObj:=FakeWing;
        MoveL Target_4890,v30,fine,DrillTool\WObj:=FakeWing;
SetDO drillDone,1;
WaitUntil drillDone = 0;
        MoveL RelTool(Target_4890,0,0,-10),v30,z10,DrillTool\WObj:=FakeWing;
        MoveL RelTool(Target_4900,0,0,-10),v30,z10,DrillTool\WObj:=FakeWing;
        MoveL Target_4900,v30,fine,DrillTool\WObj:=FakeWing;
SetDO drillDone,1;
WaitUntil drillDone = 0;
        MoveL RelTool(Target_4900,0,0,-10),v30,z10,DrillTool\WObj:=FakeWing;
        MoveL RelTool(Target_4910,0,0,-10),v30,z10,DrillTool\WObj:=FakeWing;
        MoveL Target_4910,v30,fine,DrillTool\WObj:=FakeWing;
SetDO drillDone,1;
WaitUntil drillDone = 0;
        MoveL RelTool(Target_4910,0,0,-10),v30,z10,DrillTool\WObj:=FakeWing;
        MoveL RelTool(Target_4920,0,0,-10),v30,z10,DrillTool\WObj:=FakeWing;
        MoveL Target_4920,v30,fine,DrillTool\WObj:=FakeWing;
SetDO drillDone,1;
WaitUntil drillDone = 0;
        MoveL RelTool(Target_4920,0,0,-10),v30,z10,DrillTool\WObj:=FakeWing;
        MoveL RelTool(Target_4930,0,0,-10),v30,z10,DrillTool\WObj:=FakeWing;
        MoveL Target_4930,v30,fine,DrillTool\WObj:=FakeWing;
SetDO drillDone,1;
WaitUntil drillDone = 0;
        MoveL RelTool(Target_4930,0,0,-10),v30,z10,DrillTool\WObj:=FakeWing;
        MoveL RelTool(Target_4940,0,0,-10),v30,z10,DrillTool\WObj:=FakeWing;
        MoveL Target_4940,v30,fine,DrillTool\WObj:=FakeWing;
SetDO drillDone,1;
WaitUntil drillDone = 0;
        MoveL RelTool(Target_4940,0,0,-10),v30,z10,DrillTool\WObj:=FakeWing;
        MoveL RelTool(Target_4950,0,0,-10),v30,z10,DrillTool\WObj:=FakeWing;
        MoveL Target_4950,v30,fine,DrillTool\WObj:=FakeWing;
SetDO drillDone,1;
WaitUntil drillDone = 0;
        MoveL RelTool(Target_4950,0,0,-10),v30,z10,DrillTool\WObj:=FakeWing;
        MoveL RelTool(Target_4960,0,0,-10),v30,z10,DrillTool\WObj:=FakeWing;
        MoveL Target_4960,v30,fine,DrillTool\WObj:=FakeWing;
SetDO drillDone,1;
WaitUntil drillDone = 0;
        MoveL RelTool(Target_4960,0,0,-10),v30,z10,DrillTool\WObj:=FakeWing;
        MoveL RelTool(Target_4970,0,0,-10),v30,z10,DrillTool\WObj:=FakeWing;
        MoveL Target_4970,v30,fine,DrillTool\WObj:=FakeWing;
SetDO drillDone,1;
WaitUntil drillDone = 0;
        MoveL RelTool(Target_4970,0,0,-10),v30,z10,DrillTool\WObj:=FakeWing;
        MoveL RelTool(Target_4980,0,0,-10),v30,z10,DrillTool\WObj:=FakeWing;
        MoveL Target_4980,v30,fine,DrillTool\WObj:=FakeWing;
SetDO drillDone,1;
WaitUntil drillDone = 0;
        MoveL RelTool(Target_4980,0,0,-10),v30,z10,DrillTool\WObj:=FakeWing;
        MoveL RelTool(Target_4990,0,0,-10),v30,z10,DrillTool\WObj:=FakeWing;
        MoveL Target_4990,v30,fine,DrillTool\WObj:=FakeWing;
SetDO drillDone,1;
WaitUntil drillDone = 0;
        MoveL RelTool(Target_4990,0,0,-10),v30,z10,DrillTool\WObj:=FakeWing;
        MoveL RelTool(Target_5000,0,0,-10),v30,z10,DrillTool\WObj:=FakeWing;
        MoveL Target_5000,v30,fine,DrillTool\WObj:=FakeWing;
SetDO drillDone,1;
WaitUntil drillDone = 0;
        MoveL RelTool(Target_5000,0,0,-10),v30,z10,DrillTool\WObj:=FakeWing;
        MoveL RelTool(Target_5010,0,0,-10),v30,z10,DrillTool\WObj:=FakeWing;
        MoveL Target_5010,v30,fine,DrillTool\WObj:=FakeWing;
SetDO drillDone,1;
WaitUntil drillDone = 0;
        MoveL RelTool(Target_5010,0,0,-10),v30,z10,DrillTool\WObj:=FakeWing;
        MoveL RelTool(Target_5020,0,0,-10),v30,z10,DrillTool\WObj:=FakeWing;
        MoveL Target_5020,v30,fine,DrillTool\WObj:=FakeWing;
SetDO drillDone,1;
WaitUntil drillDone = 0;
        MoveL RelTool(Target_5020,0,0,-10),v30,z10,DrillTool\WObj:=FakeWing;
        MoveL RelTool(Target_5030,0,0,-10),v30,z10,DrillTool\WObj:=FakeWing;
        MoveL Target_5030,v30,fine,DrillTool\WObj:=FakeWing;
SetDO drillDone,1;
WaitUntil drillDone = 0;
        MoveL RelTool(Target_5030,0,0,-10),v30,z10,DrillTool\WObj:=FakeWing;
        MoveL RelTool(Target_5040,0,0,-10),v30,z10,DrillTool\WObj:=FakeWing;
        MoveL Target_5040,v30,fine,DrillTool\WObj:=FakeWing;
SetDO drillDone,1;
WaitUntil drillDone = 0;
        MoveL RelTool(Target_5040,0,0,-10),v30,z10,DrillTool\WObj:=FakeWing;
        MoveL RelTool(Target_5050,0,0,-10),v30,z10,DrillTool\WObj:=FakeWing;
        MoveL Target_5050,v30,fine,DrillTool\WObj:=FakeWing;
SetDO drillDone,1;
WaitUntil drillDone = 0;
        MoveL RelTool(Target_5050,0,0,-10),v30,z10,DrillTool\WObj:=FakeWing;
        MoveL RelTool(Target_5060,0,0,-10),v30,z10,DrillTool\WObj:=FakeWing;
        MoveL Target_5060,v30,fine,DrillTool\WObj:=FakeWing;
SetDO drillDone,1;
WaitUntil drillDone = 0;
        MoveL RelTool(Target_5060,0,0,-10),v30,z10,DrillTool\WObj:=FakeWing;
        MoveL RelTool(Target_5070,0,0,-10),v30,z10,DrillTool\WObj:=FakeWing;
        MoveL Target_5070,v30,fine,DrillTool\WObj:=FakeWing;
SetDO drillDone,1;
WaitUntil drillDone = 0;
        MoveL RelTool(Target_5070,0,0,-10),v30,z10,DrillTool\WObj:=FakeWing;
        MoveL RelTool(Target_5080,0,0,-10),v30,z10,DrillTool\WObj:=FakeWing;
        MoveL Target_5080,v30,fine,DrillTool\WObj:=FakeWing;
SetDO drillDone,1;
WaitUntil drillDone = 0;
        MoveL RelTool(Target_5080,0,0,-10),v30,z10,DrillTool\WObj:=FakeWing;
        MoveL RelTool(Target_5090,0,0,-10),v30,z10,DrillTool\WObj:=FakeWing;
        MoveL Target_5090,v30,fine,DrillTool\WObj:=FakeWing;
SetDO drillDone,1;
WaitUntil drillDone = 0;
        MoveL RelTool(Target_5090,0,0,-10),v30,z10,DrillTool\WObj:=FakeWing;
        MoveL RelTool(Target_5100,0,0,-10),v30,z10,DrillTool\WObj:=FakeWing;
        MoveL Target_5100,v30,fine,DrillTool\WObj:=FakeWing;
SetDO drillDone,1;
WaitUntil drillDone = 0;
        MoveL RelTool(Target_5100,0,0,-10),v30,z10,DrillTool\WObj:=FakeWing;
        MoveL RelTool(Target_5110,0,0,-10),v30,z10,DrillTool\WObj:=FakeWing;
        MoveL Target_5110,v30,fine,DrillTool\WObj:=FakeWing;
SetDO drillDone,1;
WaitUntil drillDone = 0;
        MoveL RelTool(Target_5110,0,0,-10),v30,z10,DrillTool\WObj:=FakeWing;
        MoveL RelTool(Target_5120,0,0,-10),v30,z10,DrillTool\WObj:=FakeWing;
        MoveL Target_5120,v30,fine,DrillTool\WObj:=FakeWing;
SetDO drillDone,1;
WaitUntil drillDone = 0;
        MoveL RelTool(Target_5120,0,0,-10),v30,z10,DrillTool\WObj:=FakeWing;
        MoveL RelTool(Target_5130,0,0,-10),v30,z10,DrillTool\WObj:=FakeWing;
        MoveL Target_5130,v30,fine,DrillTool\WObj:=FakeWing;
SetDO drillDone,1;
WaitUntil drillDone = 0;
        MoveL RelTool(Target_5130,0,0,-10),v30,z10,DrillTool\WObj:=FakeWing;
        MoveL RelTool(Target_5140,0,0,-10),v30,z10,DrillTool\WObj:=FakeWing;
        MoveL Target_5140,v30,fine,DrillTool\WObj:=FakeWing;
SetDO drillDone,1;
WaitUntil drillDone = 0;
        MoveL RelTool(Target_5140,0,0,-10),v30,z10,DrillTool\WObj:=FakeWing;
        MoveL RelTool(Target_5150,0,0,-10),v30,z10,DrillTool\WObj:=FakeWing;
        MoveL Target_5150,v30,fine,DrillTool\WObj:=FakeWing;
SetDO drillDone,1;
WaitUntil drillDone = 0;
        MoveL RelTool(Target_5150,0,0,-10),v30,z10,DrillTool\WObj:=FakeWing;
        MoveL RelTool(Target_5160,0,0,-10),v30,z10,DrillTool\WObj:=FakeWing;
        MoveL Target_5160,v30,fine,DrillTool\WObj:=FakeWing;
SetDO drillDone,1;
WaitUntil drillDone = 0;
        MoveL RelTool(Target_5160,0,0,-10),v30,z10,DrillTool\WObj:=FakeWing;
        MoveL RelTool(Target_5170,0,0,-10),v30,z10,DrillTool\WObj:=FakeWing;
        MoveL Target_5170,v30,fine,DrillTool\WObj:=FakeWing;
SetDO drillDone,1;
WaitUntil drillDone = 0;
        MoveL RelTool(Target_5170,0,0,-10),v30,z10,DrillTool\WObj:=FakeWing;
        MoveL RelTool(Target_5180,0,0,-10),v30,z10,DrillTool\WObj:=FakeWing;
        MoveL Target_5180,v30,fine,DrillTool\WObj:=FakeWing;
SetDO drillDone,1;
WaitUntil drillDone = 0;
        MoveL RelTool(Target_5180,0,0,-10),v30,z10,DrillTool\WObj:=FakeWing;
        MoveL RelTool(Target_5190,0,0,-10),v30,z10,DrillTool\WObj:=FakeWing;
        MoveL Target_5190,v30,fine,DrillTool\WObj:=FakeWing;
SetDO drillDone,1;
WaitUntil drillDone = 0;
        MoveL RelTool(Target_5190,0,0,-10),v30,z10,DrillTool\WObj:=FakeWing;
        MoveL RelTool(Target_5200,0,0,-10),v30,z10,DrillTool\WObj:=FakeWing;
        MoveL Target_5200,v30,fine,DrillTool\WObj:=FakeWing;
SetDO drillDone,1;
WaitUntil drillDone = 0;
        MoveL RelTool(Target_5200,0,0,-10),v30,z10,DrillTool\WObj:=FakeWing;
        MoveL RelTool(Target_5210,0,0,-10),v30,z10,DrillTool\WObj:=FakeWing;
        MoveL Target_5210,v30,fine,DrillTool\WObj:=FakeWing;
SetDO drillDone,1;
WaitUntil drillDone = 0;
        MoveL RelTool(Target_5210,0,0,-10),v30,z10,DrillTool\WObj:=FakeWing;
        MoveL RelTool(Target_5220,0,0,-10),v30,z10,DrillTool\WObj:=FakeWing;
        MoveL Target_5220,v30,fine,DrillTool\WObj:=FakeWing;
SetDO drillDone,1;
WaitUntil drillDone = 0;
        MoveL RelTool(Target_5220,0,0,-10),v30,z10,DrillTool\WObj:=FakeWing;
        MoveL RelTool(Target_5230,0,0,-10),v30,z10,DrillTool\WObj:=FakeWing;
        MoveL Target_5230,v30,fine,DrillTool\WObj:=FakeWing;
SetDO drillDone,1;
WaitUntil drillDone = 0;
        MoveL RelTool(Target_5230,0,0,-10),v30,z10,DrillTool\WObj:=FakeWing;
        MoveL RelTool(Target_5240,0,0,-10),v30,z10,DrillTool\WObj:=FakeWing;
        MoveL Target_5240,v30,fine,DrillTool\WObj:=FakeWing;
SetDO drillDone,1;
WaitUntil drillDone = 0;
        MoveL RelTool(Target_5240,0,0,-10),v30,z10,DrillTool\WObj:=FakeWing;
        MoveL RelTool(Target_5250,0,0,-10),v30,z10,DrillTool\WObj:=FakeWing;
        MoveL Target_5250,v30,fine,DrillTool\WObj:=FakeWing;
SetDO drillDone,1;
WaitUntil drillDone = 0;
        MoveL RelTool(Target_5250,0,0,-10),v30,z10,DrillTool\WObj:=FakeWing;
        MoveL RelTool(Target_5260,0,0,-10),v30,z10,DrillTool\WObj:=FakeWing;
        MoveL Target_5260,v30,fine,DrillTool\WObj:=FakeWing;
SetDO drillDone,1;
WaitUntil drillDone = 0;
        MoveL RelTool(Target_5260,0,0,-10),v30,z10,DrillTool\WObj:=FakeWing;
        MoveL RelTool(Target_5270,0,0,-10),v30,z10,DrillTool\WObj:=FakeWing;
        MoveL Target_5270,v30,fine,DrillTool\WObj:=FakeWing;
SetDO drillDone,1;
WaitUntil drillDone = 0;
        MoveL RelTool(Target_5270,0,0,-10),v30,z10,DrillTool\WObj:=FakeWing;
        MoveL RelTool(Target_5280,0,0,-10),v30,z10,DrillTool\WObj:=FakeWing;
        MoveL Target_5280,v30,fine,DrillTool\WObj:=FakeWing;
SetDO drillDone,1;
WaitUntil drillDone = 0;
        MoveL RelTool(Target_5280,0,0,-10),v30,z10,DrillTool\WObj:=FakeWing;
        MoveL RelTool(Target_5290,0,0,-10),v30,z10,DrillTool\WObj:=FakeWing;
        MoveL Target_5290,v30,fine,DrillTool\WObj:=FakeWing;
SetDO drillDone,1;
WaitUntil drillDone = 0;
        MoveL RelTool(Target_5290,0,0,-10),v30,z10,DrillTool\WObj:=FakeWing;
        MoveL RelTool(Target_5300,0,0,-10),v30,z10,DrillTool\WObj:=FakeWing;
        MoveL Target_5300,v30,fine,DrillTool\WObj:=FakeWing;
SetDO drillDone,1;
WaitUntil drillDone = 0;
        MoveL RelTool(Target_5300,0,0,-10),v30,z10,DrillTool\WObj:=FakeWing;
        MoveL RelTool(Target_5310,0,0,-10),v30,z10,DrillTool\WObj:=FakeWing;
        MoveL Target_5310,v30,fine,DrillTool\WObj:=FakeWing;
SetDO drillDone,1;
WaitUntil drillDone = 0;
        MoveL RelTool(Target_5310,0,0,-10),v30,z10,DrillTool\WObj:=FakeWing;
        MoveL RelTool(Target_5320,0,0,-10),v30,z10,DrillTool\WObj:=FakeWing;
        MoveL Target_5320,v30,fine,DrillTool\WObj:=FakeWing;
SetDO drillDone,1;
WaitUntil drillDone = 0;
        MoveL RelTool(Target_5320,0,0,-10),v30,z10,DrillTool\WObj:=FakeWing;
        MoveL RelTool(Target_5330,0,0,-10),v30,z10,DrillTool\WObj:=FakeWing;
        MoveL Target_5330,v30,fine,DrillTool\WObj:=FakeWing;
SetDO drillDone,1;
WaitUntil drillDone = 0;
        MoveL RelTool(Target_5330,0,0,-10),v30,z10,DrillTool\WObj:=FakeWing;
        MoveL RelTool(Target_5340,0,0,-10),v30,z10,DrillTool\WObj:=FakeWing;
        MoveL Target_5340,v30,fine,DrillTool\WObj:=FakeWing;
SetDO drillDone,1;
WaitUntil drillDone = 0;
        MoveL RelTool(Target_5340,0,0,-10),v30,z10,DrillTool\WObj:=FakeWing;
        MoveL RelTool(Target_5350,0,0,-10),v30,z10,DrillTool\WObj:=FakeWing;
        MoveL Target_5350,v30,fine,DrillTool\WObj:=FakeWing;
SetDO drillDone,1;
WaitUntil drillDone = 0;
        MoveL RelTool(Target_5350,0,0,-10),v30,z10,DrillTool\WObj:=FakeWing;
        MoveL RelTool(Target_5360,0,0,-10),v30,z10,DrillTool\WObj:=FakeWing;
        MoveL Target_5360,v30,fine,DrillTool\WObj:=FakeWing;
SetDO drillDone,1;
WaitUntil drillDone = 0;
        MoveL RelTool(Target_5360,0,0,-10),v30,z10,DrillTool\WObj:=FakeWing;
        MoveL RelTool(Target_5370,0,0,-10),v30,z10,DrillTool\WObj:=FakeWing;
        MoveL Target_5370,v30,fine,DrillTool\WObj:=FakeWing;
SetDO drillDone,1;
WaitUntil drillDone = 0;
        MoveL RelTool(Target_5370,0,0,-10),v30,z10,DrillTool\WObj:=FakeWing;
        MoveL RelTool(Target_5380,0,0,-10),v30,z10,DrillTool\WObj:=FakeWing;
        MoveL Target_5380,v30,fine,DrillTool\WObj:=FakeWing;
SetDO drillDone,1;
WaitUntil drillDone = 0;
        MoveL RelTool(Target_5380,0,0,-10),v30,z10,DrillTool\WObj:=FakeWing;
        MoveL RelTool(Target_5390,0,0,-10),v30,z10,DrillTool\WObj:=FakeWing;
        MoveL Target_5390,v30,fine,DrillTool\WObj:=FakeWing;
SetDO drillDone,1;
WaitUntil drillDone = 0;
        MoveL RelTool(Target_5390,0,0,-10),v30,z10,DrillTool\WObj:=FakeWing;
        MoveL RelTool(Target_5400,0,0,-10),v30,z10,DrillTool\WObj:=FakeWing;
        MoveL Target_5400,v30,fine,DrillTool\WObj:=FakeWing;
SetDO drillDone,1;
WaitUntil drillDone = 0;
        MoveL RelTool(Target_5400,0,0,-10),v30,z10,DrillTool\WObj:=FakeWing;
        MoveL RelTool(Target_5410,0,0,-10),v30,z10,DrillTool\WObj:=FakeWing;
        MoveL Target_5410,v30,fine,DrillTool\WObj:=FakeWing;
SetDO drillDone,1;
WaitUntil drillDone = 0;
        MoveL RelTool(Target_5410,0,0,-10),v30,z10,DrillTool\WObj:=FakeWing;
        MoveL RelTool(Target_5420,0,0,-10),v30,z10,DrillTool\WObj:=FakeWing;
        MoveL Target_5420,v30,fine,DrillTool\WObj:=FakeWing;
SetDO drillDone,1;
WaitUntil drillDone = 0;
        MoveL RelTool(Target_5420,0,0,-10),v30,z10,DrillTool\WObj:=FakeWing;
        MoveL RelTool(Target_5430,0,0,-10),v30,z10,DrillTool\WObj:=FakeWing;
        MoveL Target_5430,v30,fine,DrillTool\WObj:=FakeWing;
SetDO drillDone,1;
WaitUntil drillDone = 0;
        MoveL RelTool(Target_5430,0,0,-10),v30,z10,DrillTool\WObj:=FakeWing;
        MoveL RelTool(Target_5440,0,0,-10),v30,z10,DrillTool\WObj:=FakeWing;
        MoveL Target_5440,v30,fine,DrillTool\WObj:=FakeWing;
SetDO drillDone,1;
WaitUntil drillDone = 0;
        MoveL RelTool(Target_5440,0,0,-10),v30,z10,DrillTool\WObj:=FakeWing;
        MoveL RelTool(Target_5450,0,0,-10),v30,z10,DrillTool\WObj:=FakeWing;
        MoveL Target_5450,v30,fine,DrillTool\WObj:=FakeWing;
SetDO drillDone,1;
WaitUntil drillDone = 0;
        MoveL RelTool(Target_5450,0,0,-10),v30,z10,DrillTool\WObj:=FakeWing;
        MoveL RelTool(Target_5460,0,0,-10),v30,z10,DrillTool\WObj:=FakeWing;
        MoveL Target_5460,v30,fine,DrillTool\WObj:=FakeWing;
SetDO drillDone,1;
WaitUntil drillDone = 0;
        MoveL RelTool(Target_5460,0,0,-10),v30,z10,DrillTool\WObj:=FakeWing;
        MoveL RelTool(Target_5470,0,0,-10),v30,z10,DrillTool\WObj:=FakeWing;
        MoveL Target_5470,v30,fine,DrillTool\WObj:=FakeWing;
SetDO drillDone,1;
WaitUntil drillDone = 0;
        MoveL RelTool(Target_5470,0,0,-10),v30,z10,DrillTool\WObj:=FakeWing;
        MoveL RelTool(Target_5480,0,0,-10),v30,z10,DrillTool\WObj:=FakeWing;
        MoveL Target_5480,v30,fine,DrillTool\WObj:=FakeWing;
SetDO drillDone,1;
WaitUntil drillDone = 0;
        MoveL RelTool(Target_5480,0,0,-10),v30,z10,DrillTool\WObj:=FakeWing;
        MoveL RelTool(Target_5490,0,0,-10),v30,z10,DrillTool\WObj:=FakeWing;
        MoveL Target_5490,v30,fine,DrillTool\WObj:=FakeWing;
SetDO drillDone,1;
WaitUntil drillDone = 0;
        MoveL RelTool(Target_5490,0,0,-10),v30,z10,DrillTool\WObj:=FakeWing;
        MoveL RelTool(Target_5500,0,0,-10),v30,z10,DrillTool\WObj:=FakeWing;
        MoveL Target_5500,v30,fine,DrillTool\WObj:=FakeWing;
SetDO drillDone,1;
WaitUntil drillDone = 0;
        MoveL RelTool(Target_5500,0,0,-10),v30,z10,DrillTool\WObj:=FakeWing;
        MoveL RelTool(Target_5510,0,0,-10),v30,z10,DrillTool\WObj:=FakeWing;
        MoveL Target_5510,v30,fine,DrillTool\WObj:=FakeWing;
SetDO drillDone,1;
WaitUntil drillDone = 0;
        MoveL RelTool(Target_5510,0,0,-10),v30,z10,DrillTool\WObj:=FakeWing;
        MoveL RelTool(Target_5520,0,0,-10),v30,z10,DrillTool\WObj:=FakeWing;
        MoveL Target_5520,v30,fine,DrillTool\WObj:=FakeWing;
SetDO drillDone,1;
WaitUntil drillDone = 0;
        MoveL RelTool(Target_5520,0,0,-10),v30,z10,DrillTool\WObj:=FakeWing;
        MoveL RelTool(Target_5530,0,0,-10),v30,z10,DrillTool\WObj:=FakeWing;
        MoveL Target_5530,v30,fine,DrillTool\WObj:=FakeWing;
SetDO drillDone,1;
WaitUntil drillDone = 0;
        MoveL RelTool(Target_5530,0,0,-10),v30,z10,DrillTool\WObj:=FakeWing;
        MoveL RelTool(Target_5540,0,0,-10),v30,z10,DrillTool\WObj:=FakeWing;
        MoveL Target_5540,v30,fine,DrillTool\WObj:=FakeWing;
SetDO drillDone,1;
WaitUntil drillDone = 0;
        MoveL RelTool(Target_5540,0,0,-10),v30,z10,DrillTool\WObj:=FakeWing;
        MoveL RelTool(Target_5550,0,0,-10),v30,z10,DrillTool\WObj:=FakeWing;
        MoveL Target_5550,v30,fine,DrillTool\WObj:=FakeWing;
SetDO drillDone,1;
WaitUntil drillDone = 0;
        MoveL RelTool(Target_5550,0,0,-10),v30,z10,DrillTool\WObj:=FakeWing;
        MoveL RelTool(Target_5560,0,0,-10),v30,z10,DrillTool\WObj:=FakeWing;
        MoveL Target_5560,v30,fine,DrillTool\WObj:=FakeWing;
SetDO drillDone,1;
WaitUntil drillDone = 0;
        MoveL RelTool(Target_5560,0,0,-10),v30,z10,DrillTool\WObj:=FakeWing;
        MoveL RelTool(Target_5570,0,0,-10),v30,z10,DrillTool\WObj:=FakeWing;
        MoveL Target_5570,v30,fine,DrillTool\WObj:=FakeWing;
SetDO drillDone,1;
WaitUntil drillDone = 0;
        MoveL RelTool(Target_5570,0,0,-10),v30,z10,DrillTool\WObj:=FakeWing;
        MoveL RelTool(Target_5580,0,0,-10),v30,z10,DrillTool\WObj:=FakeWing;
        MoveL Target_5580,v30,fine,DrillTool\WObj:=FakeWing;
SetDO drillDone,1;
WaitUntil drillDone = 0;
        MoveL RelTool(Target_5580,0,0,-10),v30,z10,DrillTool\WObj:=FakeWing;
        MoveL RelTool(Target_5590,0,0,-10),v30,z10,DrillTool\WObj:=FakeWing;
        MoveL Target_5590,v30,fine,DrillTool\WObj:=FakeWing;
SetDO drillDone,1;
WaitUntil drillDone = 0;
        MoveL RelTool(Target_5590,0,0,-10),v30,z10,DrillTool\WObj:=FakeWing;
        MoveL RelTool(Target_5600,0,0,-10),v30,z10,DrillTool\WObj:=FakeWing;
        MoveL Target_5600,v30,fine,DrillTool\WObj:=FakeWing;
SetDO drillDone,1;
WaitUntil drillDone = 0;
        MoveL RelTool(Target_5600,0,0,-10),v30,z10,DrillTool\WObj:=FakeWing;
        MoveL RelTool(Target_5610,0,0,-10),v30,z10,DrillTool\WObj:=FakeWing;
        MoveL Target_5610,v30,fine,DrillTool\WObj:=FakeWing;
SetDO drillDone,1;
WaitUntil drillDone = 0;
        MoveL RelTool(Target_5610,0,0,-10),v30,z10,DrillTool\WObj:=FakeWing;
        MoveL RelTool(Target_5620,0,0,-10),v30,z10,DrillTool\WObj:=FakeWing;
        MoveL Target_5620,v30,fine,DrillTool\WObj:=FakeWing;
SetDO drillDone,1;
WaitUntil drillDone = 0;
        MoveL RelTool(Target_5620,0,0,-10),v30,z10,DrillTool\WObj:=FakeWing;
        MoveL RelTool(Target_5630,0,0,-10),v30,z10,DrillTool\WObj:=FakeWing;
        MoveL Target_5630,v30,fine,DrillTool\WObj:=FakeWing;
SetDO drillDone,1;
WaitUntil drillDone = 0;
        MoveL RelTool(Target_5630,0,0,-10),v30,z10,DrillTool\WObj:=FakeWing;
        MoveL RelTool(Target_5640,0,0,-10),v30,z10,DrillTool\WObj:=FakeWing;
        MoveL Target_5640,v30,fine,DrillTool\WObj:=FakeWing;
SetDO drillDone,1;
WaitUntil drillDone = 0;
        MoveL RelTool(Target_5640,0,0,-10),v30,z10,DrillTool\WObj:=FakeWing;
        MoveL RelTool(Target_5650,0,0,-10),v30,z10,DrillTool\WObj:=FakeWing;
        MoveL Target_5650,v30,fine,DrillTool\WObj:=FakeWing;
SetDO drillDone,1;
WaitUntil drillDone = 0;
        MoveL RelTool(Target_5650,0,0,-10),v30,z10,DrillTool\WObj:=FakeWing;
        MoveL RelTool(Target_5660,0,0,-10),v30,z10,DrillTool\WObj:=FakeWing;
        MoveL Target_5660,v30,fine,DrillTool\WObj:=FakeWing;
SetDO drillDone,1;
WaitUntil drillDone = 0;
        MoveL RelTool(Target_5660,0,0,-10),v30,z10,DrillTool\WObj:=FakeWing;
        MoveL RelTool(Target_5670,0,0,-10),v30,z10,DrillTool\WObj:=FakeWing;
        MoveL Target_5670,v30,fine,DrillTool\WObj:=FakeWing;
SetDO drillDone,1;
WaitUntil drillDone = 0;
        MoveL RelTool(Target_5670,0,0,-10),v30,z10,DrillTool\WObj:=FakeWing;
        MoveL RelTool(Target_5680,0,0,-10),v30,z10,DrillTool\WObj:=FakeWing;
        MoveL Target_5680,v30,fine,DrillTool\WObj:=FakeWing;
SetDO drillDone,1;
WaitUntil drillDone = 0;
        MoveL RelTool(Target_5680,0,0,-10),v30,z10,DrillTool\WObj:=FakeWing;
        MoveL RelTool(Target_5690,0,0,-10),v30,z10,DrillTool\WObj:=FakeWing;
        MoveL Target_5690,v30,fine,DrillTool\WObj:=FakeWing;
SetDO drillDone,1;
WaitUntil drillDone = 0;
        MoveL RelTool(Target_5690,0,0,-10),v30,z10,DrillTool\WObj:=FakeWing;
        MoveL RelTool(Target_5700,0,0,-10),v30,z10,DrillTool\WObj:=FakeWing;
        MoveL Target_5700,v30,fine,DrillTool\WObj:=FakeWing;
SetDO drillDone,1;
WaitUntil drillDone = 0;
        MoveL RelTool(Target_5700,0,0,-10),v30,z10,DrillTool\WObj:=FakeWing;
        MoveL RelTool(Target_5710,0,0,-10),v30,z10,DrillTool\WObj:=FakeWing;
        MoveL Target_5710,v30,fine,DrillTool\WObj:=FakeWing;
SetDO drillDone,1;
WaitUntil drillDone = 0;
        MoveL RelTool(Target_5710,0,0,-10),v30,z10,DrillTool\WObj:=FakeWing;
        MoveL RelTool(Target_5720,0,0,-10),v30,z10,DrillTool\WObj:=FakeWing;
        MoveL Target_5720,v30,fine,DrillTool\WObj:=FakeWing;
SetDO drillDone,1;
WaitUntil drillDone = 0;
        MoveL RelTool(Target_5720,0,0,-10),v30,z10,DrillTool\WObj:=FakeWing;
        MoveL RelTool(Target_5730,0,0,-10),v30,z10,DrillTool\WObj:=FakeWing;
        MoveL Target_5730,v30,fine,DrillTool\WObj:=FakeWing;
SetDO drillDone,1;
WaitUntil drillDone = 0;
        MoveL RelTool(Target_5730,0,0,-10),v30,z10,DrillTool\WObj:=FakeWing;
        MoveL RelTool(Target_5740,0,0,-10),v30,z10,DrillTool\WObj:=FakeWing;
        MoveL Target_5740,v30,fine,DrillTool\WObj:=FakeWing;
SetDO drillDone,1;
WaitUntil drillDone = 0;
        MoveL RelTool(Target_5740,0,0,-10),v30,z10,DrillTool\WObj:=FakeWing;
        MoveL RelTool(Target_5750,0,0,-10),v30,z10,DrillTool\WObj:=FakeWing;
        MoveL Target_5750,v30,fine,DrillTool\WObj:=FakeWing;
SetDO drillDone,1;
WaitUntil drillDone = 0;
        MoveL RelTool(Target_5750,0,0,-10),v30,z10,DrillTool\WObj:=FakeWing;
        MoveL RelTool(Target_5760,0,0,-10),v30,z10,DrillTool\WObj:=FakeWing;
        MoveL Target_5760,v30,fine,DrillTool\WObj:=FakeWing;
SetDO drillDone,1;
WaitUntil drillDone = 0;
        MoveL RelTool(Target_5760,0,0,-10),v30,z10,DrillTool\WObj:=FakeWing;
        MoveL RelTool(Target_5770,0,0,-10),v30,z10,DrillTool\WObj:=FakeWing;
        MoveL Target_5770,v30,fine,DrillTool\WObj:=FakeWing;
SetDO drillDone,1;
WaitUntil drillDone = 0;
        MoveL RelTool(Target_5770,0,0,-10),v30,z10,DrillTool\WObj:=FakeWing;
        MoveL RelTool(Target_5780,0,0,-10),v30,z10,DrillTool\WObj:=FakeWing;
        MoveL Target_5780,v30,fine,DrillTool\WObj:=FakeWing;
SetDO drillDone,1;
WaitUntil drillDone = 0;
        MoveL RelTool(Target_5780,0,0,-10),v30,z10,DrillTool\WObj:=FakeWing;
        MoveL RelTool(Target_5790,0,0,-10),v30,z10,DrillTool\WObj:=FakeWing;
        MoveL Target_5790,v30,fine,DrillTool\WObj:=FakeWing;
SetDO drillDone,1;
WaitUntil drillDone = 0;
        MoveL RelTool(Target_5790,0,0,-10),v30,z10,DrillTool\WObj:=FakeWing;
        MoveL RelTool(Target_5800,0,0,-10),v30,z10,DrillTool\WObj:=FakeWing;
        MoveL Target_5800,v30,fine,DrillTool\WObj:=FakeWing;
SetDO drillDone,1;
WaitUntil drillDone = 0;
        MoveL RelTool(Target_5800,0,0,-10),v30,z10,DrillTool\WObj:=FakeWing;
        MoveL RelTool(Target_5810,0,0,-10),v30,z10,DrillTool\WObj:=FakeWing;
        MoveL Target_5810,v30,fine,DrillTool\WObj:=FakeWing;
SetDO drillDone,1;
WaitUntil drillDone = 0;
        MoveL RelTool(Target_5810,0,0,-10),v30,z10,DrillTool\WObj:=FakeWing;
        MoveL RelTool(Target_5820,0,0,-10),v30,z10,DrillTool\WObj:=FakeWing;
        MoveL Target_5820,v30,fine,DrillTool\WObj:=FakeWing;
SetDO drillDone,1;
WaitUntil drillDone = 0;
        MoveL RelTool(Target_5820,0,0,-10),v30,z10,DrillTool\WObj:=FakeWing;
        MoveL RelTool(Target_5830,0,0,-10),v30,z10,DrillTool\WObj:=FakeWing;
        MoveL Target_5830,v30,fine,DrillTool\WObj:=FakeWing;
SetDO drillDone,1;
WaitUntil drillDone = 0;
        MoveL RelTool(Target_5830,0,0,-10),v30,z10,DrillTool\WObj:=FakeWing;
        MoveL RelTool(Target_5840,0,0,-10),v30,z10,DrillTool\WObj:=FakeWing;
        MoveL Target_5840,v30,fine,DrillTool\WObj:=FakeWing;
SetDO drillDone,1;
WaitUntil drillDone = 0;
        MoveL RelTool(Target_5840,0,0,-10),v30,z10,DrillTool\WObj:=FakeWing;
        MoveL RelTool(Target_5850,0,0,-10),v30,z10,DrillTool\WObj:=FakeWing;
        MoveL Target_5850,v30,fine,DrillTool\WObj:=FakeWing;
SetDO drillDone,1;
WaitUntil drillDone = 0;
        MoveL RelTool(Target_5850,0,0,-10),v30,z10,DrillTool\WObj:=FakeWing;
        MoveL RelTool(Target_5860,0,0,-10),v30,z10,DrillTool\WObj:=FakeWing;
        MoveL Target_5860,v30,fine,DrillTool\WObj:=FakeWing;
SetDO drillDone,1;
WaitUntil drillDone = 0;
        MoveL RelTool(Target_5860,0,0,-10),v30,z10,DrillTool\WObj:=FakeWing;
        MoveL RelTool(Target_5870,0,0,-10),v30,z10,DrillTool\WObj:=FakeWing;
        MoveL Target_5870,v30,fine,DrillTool\WObj:=FakeWing;
SetDO drillDone,1;
WaitUntil drillDone = 0;
        MoveL RelTool(Target_5870,0,0,-10),v30,z10,DrillTool\WObj:=FakeWing;
        MoveL RelTool(Target_5880,0,0,-10),v30,z10,DrillTool\WObj:=FakeWing;
        MoveL Target_5880,v30,fine,DrillTool\WObj:=FakeWing;
SetDO drillDone,1;
WaitUntil drillDone = 0;
        MoveL RelTool(Target_5880,0,0,-10),v30,z10,DrillTool\WObj:=FakeWing;
        MoveL RelTool(Target_5890,0,0,-10),v30,z10,DrillTool\WObj:=FakeWing;
        MoveL Target_5890,v30,fine,DrillTool\WObj:=FakeWing;
SetDO drillDone,1;
WaitUntil drillDone = 0;
        MoveL RelTool(Target_5890,0,0,-10),v30,z10,DrillTool\WObj:=FakeWing;
        MoveL RelTool(Target_5900,0,0,-10),v30,z10,DrillTool\WObj:=FakeWing;
        MoveL Target_5900,v30,fine,DrillTool\WObj:=FakeWing;
SetDO drillDone,1;
WaitUntil drillDone = 0;
        MoveL RelTool(Target_5900,0,0,-10),v30,z10,DrillTool\WObj:=FakeWing;
        MoveL RelTool(Target_5910,0,0,-10),v30,z10,DrillTool\WObj:=FakeWing;
        MoveL Target_5910,v30,fine,DrillTool\WObj:=FakeWing;
SetDO drillDone,1;
WaitUntil drillDone = 0;
        MoveL RelTool(Target_5910,0,0,-10),v30,z10,DrillTool\WObj:=FakeWing;
        MoveL RelTool(Target_5920,0,0,-10),v30,z10,DrillTool\WObj:=FakeWing;
        MoveL Target_5920,v30,fine,DrillTool\WObj:=FakeWing;
SetDO drillDone,1;
WaitUntil drillDone = 0;
        MoveL RelTool(Target_5920,0,0,-10),v30,z10,DrillTool\WObj:=FakeWing;
        MoveL RelTool(Target_5930,0,0,-10),v30,z10,DrillTool\WObj:=FakeWing;
        MoveL Target_5930,v30,fine,DrillTool\WObj:=FakeWing;
SetDO drillDone,1;
WaitUntil drillDone = 0;
        MoveL RelTool(Target_5930,0,0,-10),v30,z10,DrillTool\WObj:=FakeWing;
      ENDPROC
ENDMODULE

--- Backups/Rob1/SYSPAR/EIO.cfg ---
EIO:CFG_1.0:6:1::
#
EIO_SIGNAL:

      -Name "IsSuccess" -SignalType "DO" -Device "PANEL" -Label "doIsSuccess"\
      -DeviceMap "32" -Category "Virtual"

      -Name "IsComplete" -SignalType "DO" -Device "DRV_1" -Label "IsCompete"\
      -DeviceMap "33"

      -Name "IsDone" -SignalType "DO" -Label "IsDone"

--- Backups/Rob2/SYSPAR/EIO.cfg ---
EIO:CFG_1.0:6:1::
#
EIO_SIGNAL:

      -Name "doIsComplete" -SignalType "DO"
